// TIA Portal V16 export
// export: Created 2021-08-30T13:41:02.1928572Z, ExportSetting WithDefaults, DisplayName Totally Integrated Automation Portal, DisplayVersion V16 Update 3, DisplayName TIA Portal Version Control Interface, DisplayVersion V16 Update 2, DisplayName TIA Portal Openness, DisplayVersion V16 Update 3, DisplayName TIA Portal Teamcenter Gateway, DisplayVersion V16, DisplayName STEP 7 Professional, DisplayVersion V16 Update 3, DisplayName STEP 7 Safety, DisplayVersion V16, DisplayName WinCC Advanced, DisplayVersion V16 Update 3
TYPE "PropDosing"
// stored: IsFailsafeCompliant false
   STRUCT
      FE : Real;   // расход для определения дозы
      max : Real;   // доза при 20 мА
      spAuto { S7_SetPoint := 'True'} : Real := 5.0;   // задание авто (г/м3)
      spHand { S7_SetPoint := 'True'} : Real;   // задание ручное (л/ч)
      outSP : Real;   // Производительность (%)
      outPQW : Int;   // Выход на PQW
      outLPH : Real;   // Выход (л/ч)
      mode : Bool;   // 0-ручной,1-авто
      enableFix { ExternalVisible := 'False'; ExternalWritable := 'False'} : Bool;   // включение фиксированного задания
      density { S7_SetPoint := 'True'} : Real;
      outmA : Real;
      minFE { S7_SetPoint := 'True'} : Real;
      fixSP { ExternalVisible := 'False'; ExternalWritable := 'False'} : Real;   // задание от пид регулятора
      spareDint : DInt;
   END_STRUCT;
END_TYPE
